Universal Robots URScript: script_line_118.script

def script_line_118():
  set_standard_analog_input_domain(0, 1)
  set_standard_analog_input_domain(1, 1)
  set_tool_analog_input_domain(0, 1)
  set_tool_analog_input_domain(1, 1)
  set_analog_outputdomain(0, 1)
  set_analog_outputdomain(1, 1)
  set_tool_voltage(24)
  set_standard_digital_input_action(0, "default")
  set_standard_digital_input_action(1, "default")
  set_standard_digital_input_action(2, "default")
  set_standard_digital_input_action(3, "default")
  set_standard_digital_input_action(4, "default")
  set_standard_digital_input_action(5, "default")
  set_standard_digital_input_action(6, "default")
  set_standard_digital_input_action(7, "default")
  set_tool_digital_input_action(0, "default")
  set_tool_digital_input_action(1, "default")
  set_tcp(p[0.0,0.0,0.0,0.0,0.0,0.0])
  set_payload(0.0)
  set_gravity([0.0, 0.0, 9.82])
  global i_var_1=1
  global count=1
  global u26426u24231=p[0.0,0.0,0.0,0.0,0.0,0.0]
  global u24037u20855=get_forward_kin()
  while (True):
    $ 1 "机器人程序"
    $ 2 "set_digital_out(4,True)"
    set_digital_out(4,True)
    $ 3 "等待: 0.5"
    sleep(0.5)
    $ 4 "set_digital_out(4,False)"
    set_digital_out(4,False)
    $ 5 "等待: 0.5"
    sleep(0.5)
  end
end
